// TIA Portal V20 export
DATA_BLOCK "TestVarMortorstarter"   // DB223
// stored: MemoryReserve 100
   VAR
      TestplantIdentifier : WString[24] := WSTRING#'++0.000MS1';
      faceplateType : USInt;   // Bit for showing the buttons on FP
      operatorTripReset : Bool;   // Operator Trip Reset Motorstarter
      contactorControlOn { S7_SetPoint := 'True'} : Bool;
   END_VAR
BEGIN
END_DATA_BLOCK
